// TIA Portal project "practica 23" (V15)

(* hardware
DEVICE "S7-1200 station_1"  S7-1200 Station
   slot 0: "Rack_0"  S7-1200 Rack  Rack  V1.0
   slot 1: "PLC_1"  CPU 1214C AC/DC/Rly  6ES7 214-1BG40-0XB0  V4.2
   slot 101: "RF120C_1"  RF120C  6GT2 002-0LA00  V1.0
DEVICE "HMI_1"  KTP700 Basic PN
   slot 0: "HMI_1"  KTP700 Basic PN  6AV2 123-2GB03-0AX0  15.0.0.0
   slot 1: "HMI_RT_1"  KTP700 Basic PN  6AV2 123-2GB03-0AX0  15.0.0.0
   slot 5: "HMI_1.IE_CP_1"  PROFINET Interface  15.0.0.0
      slot 1: "Interfaz PROFINET_1"  PROFINET Interface
         slot 1: "Port_1"  Port
*)

// ===== PLC "PLC_1"  CPU 1214C AC/DC/Rly =====

VAR_GLOBAL   // PLC tag table "Tabla de variables estándar"
   "System_Byte" AT %MB254 : Byte;
   "FirstScan" AT %M254.0 : Bool;
   "DiagStatusUpdate" AT %M254.1 : Bool;
   "AlwaysTRUE" AT %M254.2 : Bool;
   "AlwaysFALSE" AT %M254.3 : Bool;
   "Clock_Byte" AT %MB255 : Byte;
   "Clock_10Hz" AT %M255.0 : Bool;
   "Clock_5Hz" AT %M255.1 : Bool;
   "Clock_2.5Hz" AT %M255.2 : Bool;
   "Clock_2Hz" AT %M255.3 : Bool;
   "Clock_1.25Hz" AT %M255.4 : Bool;
   "Clock_1Hz" AT %M255.5 : Bool;
   "Clock_0.625Hz" AT %M255.6 : Bool;
   "Clock_0.5Hz" AT %M255.7 : Bool;
   "boton lectura" AT %M10.0 : Bool;
   "boton escritura" AT %M10.1 : Bool;
END_VAR

DATA_BLOCK "Datos_lectura/escritura"   // DB4
{ S7_Optimized_Access := 'TRUE' }
VERSION : 0.1
   VAR
      "Datos lectura" : Array[1..1024] of Byte;
      "Datos escritura" : Array[1..1024] of Byte;
   END_VAR
BEGIN
END_DATA_BLOCK

DATA_BLOCK "Datos  HMI"   // DB6
{ S7_Optimized_Access := 'TRUE' }
VERSION : 0.1
   VAR
      "string lectura" : String;
      "string escritura" : String;
      contador : UInt;
   END_VAR
BEGIN
END_DATA_BLOCK

DATA_BLOCK "SIMATIC Ident_1"   // DB1
{ S7_Optimized_Access := 'TRUE' }
AUTHOR : SIMATIC
FAMILY : Ident
VERSION : 1.0
// stored: InstanceOfName TO_IDENT
"TO_IDENT"
BEGIN
   HW_ID := 16#010D;
   CM_CHANNEL := 1;
   LADDR := 16#0002;
END_DATA_BLOCK

ORGANIZATION_BLOCK "Main"   // OB1, LAD, ProgramCycle
TITLE = "Main Program Sweep (Cycle)"
{ S7_Optimized_Access := 'TRUE' }
VERSION : 0.1
   VAR_INPUT
      Initial_Call : Bool;   // Initial call of this OB
      Remanence : Bool;   // =True, if remanent data are available
   END_VAR
BEGIN

REGION Network 1
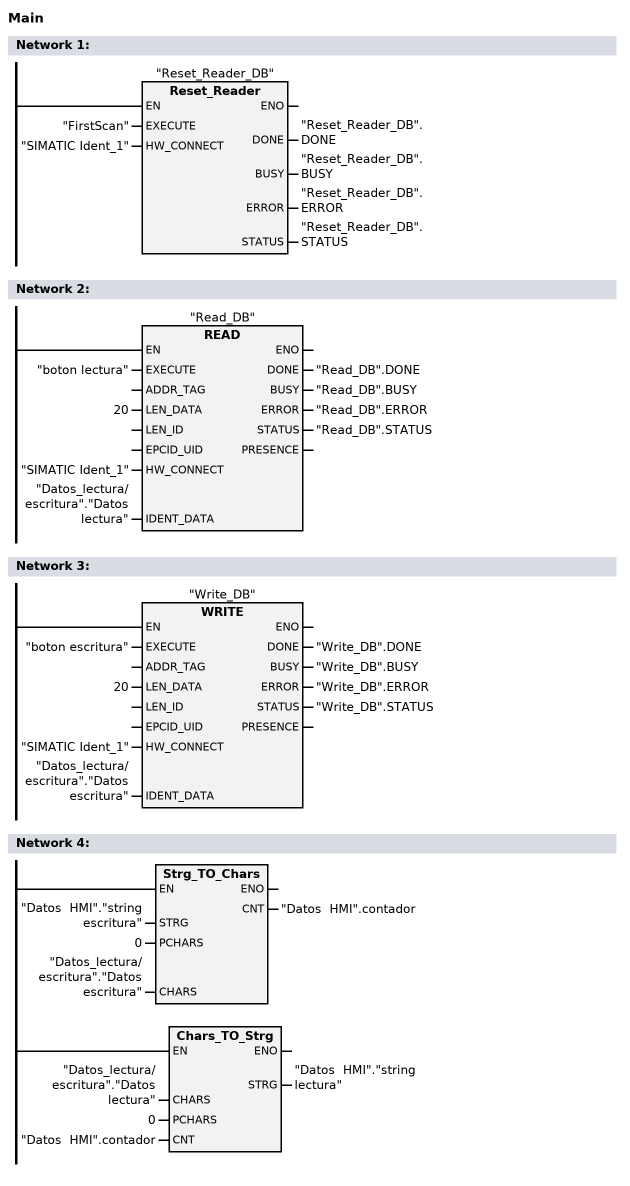
   "Reset_Reader_DB"(EXECUTE := "FirstScan",   // Reset_Reader
                     HW_CONNECT := "SIMATIC Ident_1",
                     DONE => "Reset_Reader_DB".DONE,
                     BUSY => "Reset_Reader_DB".BUSY,
                     ERROR => "Reset_Reader_DB".ERROR,
                     STATUS => "Reset_Reader_DB".STATUS);
END_REGION

REGION Network 2
   "Read_DB"(EXECUTE := "boton lectura",   // Read
             LEN_DATA := 20,
             HW_CONNECT := "SIMATIC Ident_1",
             IDENT_DATA := "Datos_lectura/escritura"."Datos lectura",
             DONE => "Read_DB".DONE,
             BUSY => "Read_DB".BUSY,
             ERROR => "Read_DB".ERROR,
             STATUS => "Read_DB".STATUS);
END_REGION

REGION Network 3
   "Write_DB"(EXECUTE := "boton escritura",   // Write
              LEN_DATA := 20,
              HW_CONNECT := "SIMATIC Ident_1",
              IDENT_DATA := "Datos_lectura/escritura"."Datos escritura",
              DONE => "Write_DB".DONE,
              BUSY => "Write_DB".BUSY,
              ERROR => "Write_DB".ERROR,
              STATUS => "Write_DB".STATUS);
END_REGION

REGION Network 4
   // no SCL statement known for Chars_TO_Strg, Strg_TO_Chars: written as a call
   Strg_TO_Chars(Strg := "Datos  HMI"."string escritura",
                 pChars := 0,
                 Chars := "Datos_lectura/escritura"."Datos escritura",
                 Cnt => "Datos  HMI".contador);
   Chars_TO_Strg(Chars := "Datos_lectura/escritura"."Datos lectura",
                 pChars := 0,
                 Cnt := "Datos  HMI".contador,
                 Strg => "Datos  HMI"."string lectura");
END_REGION
END_ORGANIZATION_BLOCK

(* ===== HMI "HMI_RT_1" =====
system functions are stored by id; their names below are inferred from use
connection "HMI_Conexión_1": ETHERNET, SMART_S7_1200_OMS

HMI tags "Tabla de variables estándar"
   "Número_imagen_variable" : UInt, internal
   "Datos recogidos de HMI_string lectura" : String[254] = PLC "Datos  HMI"."string lectura", 1 s
   "Datos recogidos de HMI_string escritura" : String[254] = PLC "Datos  HMI"."string escritura", 1 s
   "boton lectura" : Bool = PLC "boton lectura" AT %M10.0, 1 s
   "boton escritura" : Bool = PLC "boton escritura" AT %M10.1, 1 s

text list "Nombre_imagen_lista_texto": 1 'Imagen raíz'

Template "Plantilla_1" 800x480
   Button "Salir" at 714,429 size 71x50; TextOff 'Salir'; PictureOff "ExitRuntime_KTP700_Basic_PN_TR"; PictureOn "ExitRuntime_KTP700_Basic_PN_TR"
      on Release: StopRuntime(0)
   Button "Template_Button" at 614,429 size 71x50; TextOff 'Text'
   Button "Template_Button_1" at 514,429 size 71x50; TextOff 'Text'
   Button "Template_Button_2" at 414,429 size 71x50; TextOff 'Text'
   Button "Template_Button_3" at 314,429 size 71x50; TextOff 'Text'
   Button "Template_Button_4" at 214,429 size 71x50; TextOff 'Text'
   Button "Avisos" at 114,429 size 71x50; TextOff 'Avisos'; PictureOff "AlarmDisplay_KTP700_Basic_PN_TR"; PictureOn "AlarmDisplay_KTP700_Basic_PN_TR"
      on Release: function_ef3f5d25("Ventana de avisos_no_acusado", -1)
   Button "Imagen inicial" at 14,429 size 71x50; TextOff 'Imagen inicial'; PictureOff "NavigateHome_KTP700_Basic_PN_TR"; PictureOn "NavigateHome_KTP700_Basic_PN_TR"
      on Release: ActivateScreen("Imagen raíz", 0)
   SymbolicIOField "Imagen_campo_ES_simbólico" at 93,9 size 600x33; TextOff '0'; TextOn '1'; TextList "Nombre_imagen_lista_texto"
      ProcessValue <- "Número_imagen_variable"
      on Change: ActivateScreenByNumber("Número_imagen_variable", 0)
   DateTimeField "HmiScreenItemData" at 695,25 size 105x25
   DateTimeField "HmiScreenItemData_1" at 695,0 size 105x25
   GraphicView "Logotipo" at 0,0 size 91x51; Picture "Logotipo de HMI_1"

screen "Imagen raíz" 800x480, template "Plantilla_1"
   on GenerateScreen: SetBit("boton lectura")
   IOField "Campo ES_1" at 507,141 size 106x37; FormatPattern ????????????????????
      ProcessValue <- "Datos recogidos de HMI_string lectura"
   Button "Botón_1" at 507,229 size 110x46; TextOff 'Leer'
      on Press: SetBit("boton lectura")
   IOField "Campo ES_2" at 179,138 size 117x40; FormatPattern ????????????????????
      ProcessValue <- "Datos recogidos de HMI_string escritura"
   Button "Botón_2" at 178,228 size 118x47; TextOff 'Escribir'
      on Press: SetBit("boton escritura")
*)